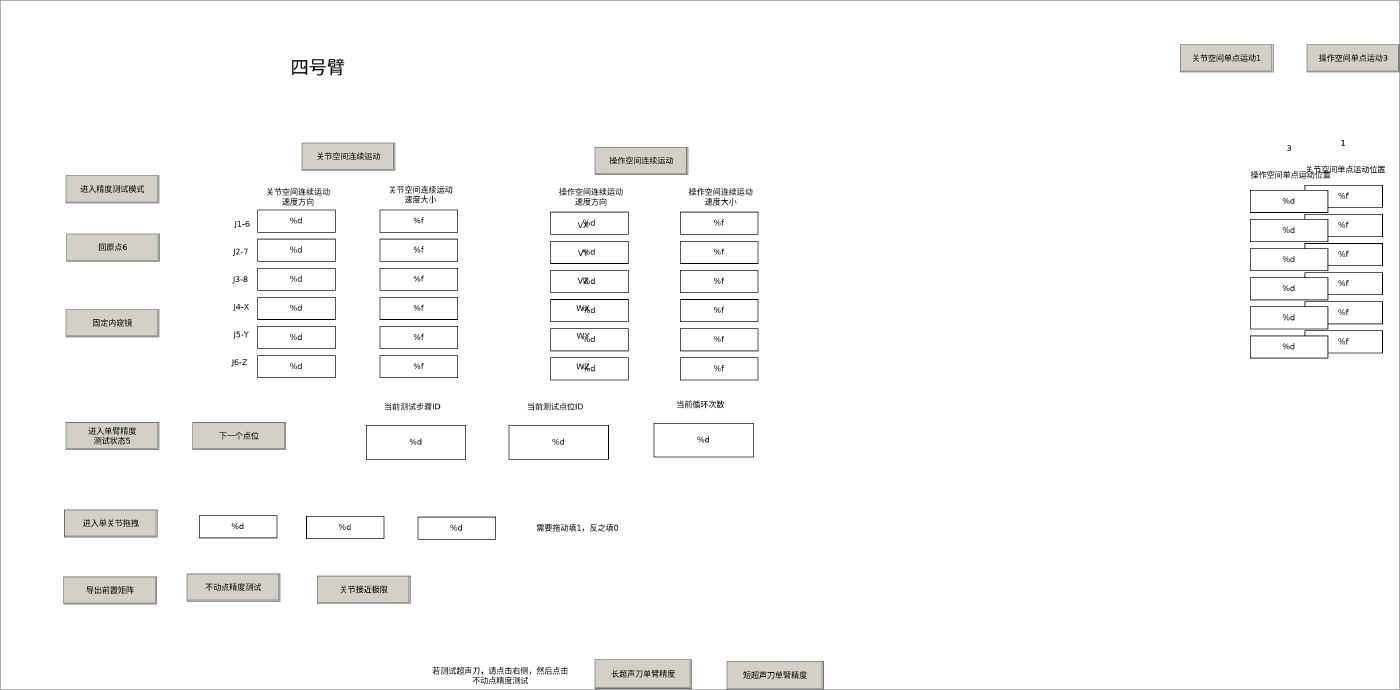
VISUALIZATION precision_a4  // 1921x948
    Button (90,241 128x38), "进入精度测试模式", colour toggle: g_motionTest.m_enterPrecisionTestMode[4]
        toggle g_motionTest.m_enterPrecisionTestMode[4]
    Label (361,71 150x43), "四号臂"
    Group (1619,61 302x38), invisible if: TRUE
        Button (0,0 128x38), "关节空间单点运动1", colour toggle: g_motionTest.m_uiArmModeL[4,1]
            tap g_motionTest.m_uiArmMode[4,1]
        Button (174,0 128x38), "操作空间单点运动3", colour toggle: g_motionTest.m_uiArmModeL[4,3]
            tap g_motionTest.m_uiArmMode[4,3]
    Button (414,196 128x38), "关节空间连续运动", colour toggle: g_motionTest.m_uiArmModeL[4,2]
        tap g_motionTest.m_uiArmMode[4,2]
    Button (816,202 128x38), "操作空间连续运动", colour toggle: g_motionTest.m_uiArmModeL[4,4]
        tap g_motionTest.m_uiArmMode[4,4]
    Button (91,321 128x38), "回原点6", colour toggle: g_motionTest.m_uiArmModeL[4,6]
        tap g_motionTest.m_uiArmMode[4,6]
    Rectangle (353,288 107x31), "%d", text variable: g_motionTest.m_jntMotionDir[4][1]
        OnMouseClick: write the text variable via Default, min -1, max 1
    Label (334,256 150x29), "关节空间连续运动 速度方向"
    Rectangle (353,328 107x31), "%d", text variable: g_motionTest.m_jntMotionDir[4][2]
        OnMouseClick: write the text variable via Default, min -1, max 1
    Rectangle (353,368 107x31), "%d", text variable: g_motionTest.m_jntMotionDir[4][3]
        OnMouseClick: write the text variable via Default, min -1, max 1
    Rectangle (353,408 107x31), "%d", text variable: g_motionTest.m_jntMotionDir[4][4]
        OnMouseClick: write the text variable via Default, min -1, max 1
    Rectangle (353,448 107x31), "%d", text variable: g_motionTest.m_jntMotionDir[4][5]
        OnMouseClick: write the text variable via Default, min -1, max 1
    Rectangle (353,488 107x31), "%d", text variable: g_motionTest.m_jntMotionDir[4][6]
        OnMouseClick: write the text variable via Default, min -1, max 1
    Group (1768,182 153x303), invisible if: TRUE
        Rectangle (22,72 107x31), "%f", text variable: g_motionTest.m_targetJntPos[4][1]
            OnMouseClick: write the text variable via Default
        Label (3,36 150x30), "关节空间单点运动位置"
        Rectangle (22,112 107x31), "%f", text variable: g_motionTest.m_targetJntPos[4][2]
            OnMouseClick: write the text variable via Default
        Rectangle (22,152 107x31), "%f", text variable: g_motionTest.m_targetJntPos[4][3]
            OnMouseClick: write the text variable via Default
        Rectangle (22,192 107x31), "%f", text variable: g_motionTest.m_targetJntPos[4][4]
            OnMouseClick: write the text variable via Default
        Rectangle (22,232 107x31), "%f", text variable: g_motionTest.m_targetJntPos[4][5]
            OnMouseClick: write the text variable via Default
        Rectangle (22,272 107x31), "%f", text variable: g_motionTest.m_targetJntPos[4][6]
            OnMouseClick: write the text variable via Default
        Label (0,0 150x30), "1"
    Rectangle (521,288 107x31), "%f", text variable: g_motionTest.m_jntVel[4][1]
        OnMouseClick: write the text variable via Default
    Label (502,253 150x29), "关节空间连续运动 速度大小"
    Rectangle (521,328 107x31), "%f", text variable: g_motionTest.m_jntVel[4][2]
        OnMouseClick: write the text variable via Default
    Rectangle (521,368 107x31), "%f", text variable: g_motionTest.m_jntVel[4][3]
        OnMouseClick: write the text variable via Default
    Rectangle (521,408 107x31), "%f", text variable: g_motionTest.m_jntVel[4][4]
        OnMouseClick: write the text variable via Default
    Rectangle (521,448 107x31), "%f", text variable: g_motionTest.m_jntVel[4][5]
        OnMouseClick: write the text variable via Default
    Rectangle (521,488 107x31), "%f", text variable: g_motionTest.m_jntVel[4][6]
        OnMouseClick: write the text variable via Default
    Group (1694,189 152x303), invisible if: TRUE
        Rectangle (21,72 107x31), "%d"
        Label (2,37 150x29), "操作空间单点运动位置"
        Rectangle (21,112 107x31), "%d"
        Rectangle (21,152 107x31), "%d"
        Rectangle (21,192 107x31), "%d"
        Rectangle (21,232 107x31), "%d"
        Rectangle (21,272 107x31), "%d"
        Label (0,0 150x30), "3"
    Rectangle (755,291 107x31), "%d", text variable: g_motionTest.m_spatialMotionDir[4][1]
        OnMouseClick: write the text variable via Default, min -1, max 1
    Label (736,256 150x29), "操作空间连续运动 速度方向"
    Rectangle (755,331 107x31), "%d", text variable: g_motionTest.m_spatialMotionDir[4][2]
        OnMouseClick: write the text variable via Default, min -1, max 1
    Rectangle (755,371 107x31), "%d", text variable: g_motionTest.m_spatialMotionDir[4][3]
        OnMouseClick: write the text variable via Default, min -1, max 1
    Rectangle (755,411 107x31), "%d", text variable: g_motionTest.m_spatialMotionDir[4][4]
        OnMouseClick: write the text variable via Default, min -1, max 1
    Rectangle (755,451 107x31), "%d", text variable: g_motionTest.m_spatialMotionDir[4][5]
        OnMouseClick: write the text variable via Default, min -1, max 1
    Rectangle (755,491 107x31), "%d", text variable: g_motionTest.m_spatialMotionDir[4][6]
        OnMouseClick: write the text variable via Default, min -1, max 1
    Rectangle (933,291 107x31), "%f", text variable: g_motionTest.m_spatialVel[4][1]
        OnMouseClick: write the text variable via Default
    Label (914,256 150x29), "操作空间连续运动 速度大小"
    Rectangle (933,331 107x31), "%f", text variable: g_motionTest.m_spatialVel[4][2]
        OnMouseClick: write the text variable via Default
    Rectangle (933,371 107x31), "%f", text variable: g_motionTest.m_spatialVel[4][3]
        OnMouseClick: write the text variable via Default
    Rectangle (933,411 107x31), "%f", text variable: g_motionTest.m_spatialVel[4][4]
        OnMouseClick: write the text variable via Default
    Rectangle (933,451 107x31), "%f", text variable: g_motionTest.m_spatialVel[4][5]
        OnMouseClick: write the text variable via Default
    Rectangle (933,491 107x31), "%f", text variable: g_motionTest.m_spatialVel[4][6]
        OnMouseClick: write the text variable via Default
    Button (90,580 128x38), "进入单臂精度 测试状态5", colour toggle: g_motionTest.m_uiArmMode[4,5]
        toggle g_motionTest.m_uiArmMode[4,5]
    Button (264,580 128x38), "下一个点位", colour toggle: g_motionTest.m_nextStep[4]
        tap g_motionTest.m_nextStep[4]
    Group (491,541 545x90)
        Rectangle (11,43 137x47), "%d", text variable: g_motionTest.m_curStep[4]
        Label (0,3 150x30), "当前测试步骤ID"
        Rectangle (207,43 137x47), "%d", text variable: g_motionTest.m_testPointId[4]
        Label (196,3 150x30), "当前测试点位ID"
        Rectangle (406,40 137x47), "%d", text variable: g_motionTest.m_testCycleId[4]
        Label (395,0 150x30), "当前循环次数"
    Group (725,295 26x224)
        Label (0,0 150x30), "VX"
        Label (0,38 150x30), "VY"
        Label (0,76 150x30), "VZ"
        Label (0,114 150x30), "WX"
        Label (0,152 150x30), "WY"
        Label (0,194 150x30), "WZ"
    Rectangle (273,708 107x31), "%d", text variable: g_motionTest.m_dragJntFlag[4][1]
        OnMouseClick: write the text variable via Default, min -1, max 1
    Button (88,700 128x38), "进入单关节拖拽", colour toggle: g_motionTest.m_uiArmMode[4,7]
        toggle g_motionTest.m_uiArmMode[4,7]
    Rectangle (420,709 107x31), "%d", text variable: g_motionTest.m_dragJntFlag[4][2]
        OnMouseClick: write the text variable via Default, min -1, max 1
    Rectangle (573,710 107x31), "%d", text variable: g_motionTest.m_dragJntFlag[4][3]
        OnMouseClick: write the text variable via Default, min -1, max 1
    Label (709,711 167x29), "需要拖动填1，反之填0"
    Button (256,788 128x38), "不动点精度测试", colour toggle: g_motionTest.m_uiArmMode[4,8]
        toggle g_motionTest.m_uiArmMode[4,8]
    Button (87,792 128x38), "导出前置矩阵"
        tap g_motionTest.m_writeData[4]
    Label (317,293 31x30), "J1-6"
    Label (307,331 47x30), "J2-7"
    Label (312,369 36x30), "J3-8"
    Label (311,407 41x30), "J4-X"
    Label (311,445 40x30), "J5-Y"
    Label (311,483 36x30), "J6-Z"
    Button (435,791 128x38), "关节接近极限", colour toggle: g_motionTest.m_jntOutFlag[4]
    Button (816,906 133x40), "长超声刀单臂精度", colour toggle: g_motionTest.m_UltrasoundKnife_Long[4]
        toggle g_motionTest.m_UltrasoundKnife_Long[4]
    Button (997,908 133x40), "短超声刀单臂精度", colour toggle: g_motionTest.m_UltrasoundKnife_Short[4]
        toggle g_motionTest.m_UltrasoundKnife_Short[4]
    Label (587,914 199x29), "若测试超声刀，请点击右侧，然后点击不动点精度测试"
    Button (90,425 128x38), "固定内窥镜", colour toggle: g_motionTest.m_uiFixedEndoFlag
        toggle g_motionTest.m_uiFixedEndoFlag
END_VISUALIZATION

(* stored: Version 1.1.0.1, ProductVersion 3.1.4024.11
   Visu precision_a4: Id {aeaf9964-9823-479c-815c-e9ce5a32a76c} *)
